(* PLC project Test, Lolitech PLCOpenEditorExample 1.0 *)
(* stored: creationDateTime 2006-09-07 18:52:43 *)

FUNCTION FBDTest : BOOL
  VAR_INPUT
    IN1 : BOOL := false;
    IN2 : BOOL := [4, [0, 1]];
    IN3 : BOOL;
  END_VAR
  VAR  (* added by the conversion: wires and edge detectors of the diagram *)
    R_TRIG1 : R_TRIG;
  END_VAR

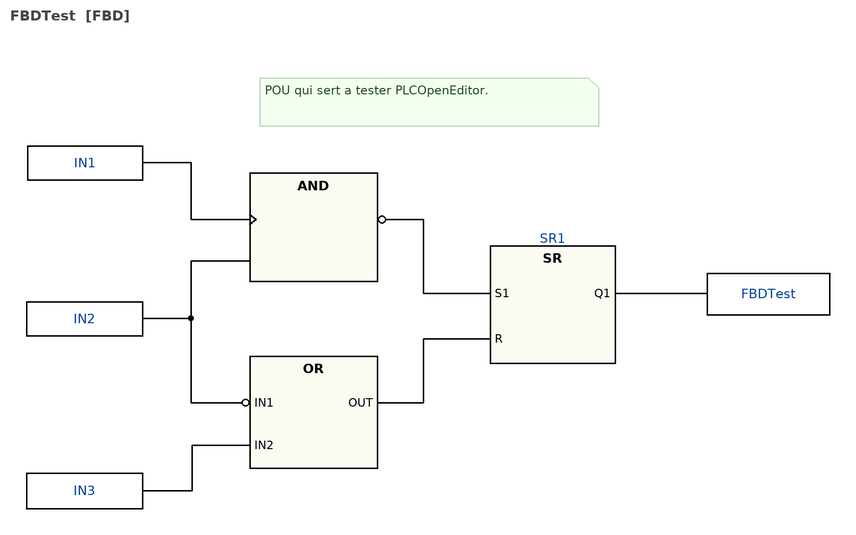
(* FBD diagram, written out as Structured Text *)
(* POU qui sert a tester PLCOpenEditor. *)
R_TRIG1(CLK := IN1);
SR1(S1 := NOT (R_TRIG1.Q AND IN2), R := NOT IN2 OR IN3);
FBDTest := SR1.Q1;
END_FUNCTION

FUNCTION LDTest : BOOL
  VAR_INPUT
    IN1 : BOOL;
    IN2 : BOOL;
    IN3 : BOOL;
    IN4 : BOOL;
  END_VAR

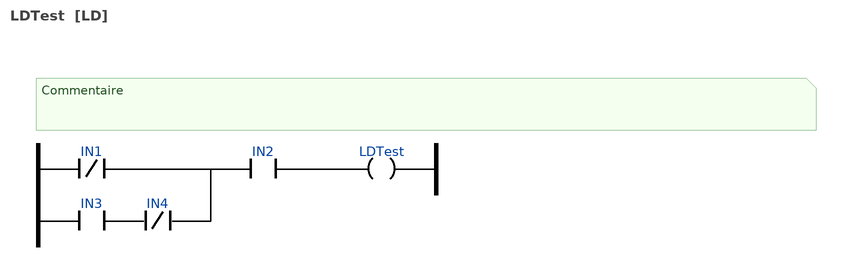
(* LD diagram, written out as Structured Text *)
(* Commentaire *)
LDTest := (NOT IN1 OR IN3 AND NOT IN4) AND IN2;
END_FUNCTION

FUNCTION ILTest : REAL
  VAR_INPUT
    X1 : REAL;
  END_VAR
  VAR
    Temp : REAL;
  END_VAR
  VAR_INPUT
    X2 : REAL;
    Y1 : REAL;
    Y2 : REAL;
    TMax : REAL;
  END_VAR
  VAR_OUTPUT
    ENO : BOOL;
  END_VAR

LD   Y1
SUB  Y2     (* Substract Y2 from Y1 *)
ST   Temp   (* Store Y1-Y2 in Temp *)
MUL  Temp   (* Multiply by Temp to square *)
ADD( X1     (* Defer ADD *)
SUB  X2     (* Substract X1 from X2 *)
ST   Temp   (* Store X1-X2 in Temp *)
MUL  Temp   (* Multiply by Temp to square *)
)
CAL  SQRT   (* Call Square root fun *)
ST   ILTest (* Setup function result *)
GT   TMax   (* Greater than TMax ? *)
JMPC ERR    (* Yes, Jump to Error *)
S    ENO    (* Set ENO *)
RET         (* Normal return *)

ERR:
RET         (* Error return, ENO not set *)
          
END_FUNCTION

PROGRAM SFCTest
  VAR_INPUT
    IN1 : BOOL;
    IN2 : BOOL;
    IN3 : BOOL;
    IN4 : BOOL;
    IN5 : BOOL;
  END_VAR

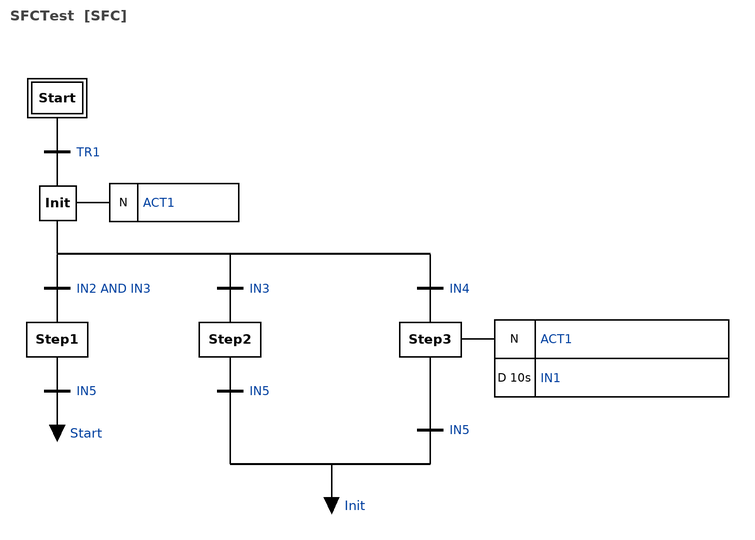
INITIAL_STEP Start:
END_STEP
TRANSITION FROM Start TO Init  (* TR1 *)
  := AND(IN1, IN2, IN3);
END_TRANSITION
STEP Init:
  ACT1(N);
END_STEP
TRANSITION FROM Init TO Step1
  := IN2 AND IN3;
END_TRANSITION
TRANSITION FROM Init TO Step2
  := IN3;
END_TRANSITION
TRANSITION FROM Init TO Step3
  := IN4;
END_TRANSITION
STEP Step1:
END_STEP
TRANSITION FROM Step1 TO Start
  := IN5;
END_TRANSITION
STEP Step2:
END_STEP
TRANSITION FROM Step2 TO Init
  := IN5;
END_TRANSITION
STEP Step3:
  ACT1(N, IN5);
  IN1(D, 10s);
END_STEP
TRANSITION FROM Step3 TO Init
  := IN5;
END_TRANSITION

ACTION ACT1:
IF IN1 THEN
	IN2 := 1;
ELSE
	IN3 := 1;
END_IF;
              
END_ACTION
END_PROGRAM

FUNCTION_BLOCK STTest
  VAR_INPUT
    Collision : BOOL;
    Gate : BOOL;
    Pump : BOOL;
    Temp : INT;
  END_VAR
  VAR_OUTPUT
    Speed : INT;
    PumpSpeed : INT;
    Brakes : BOOL;
    Control_State : BOOL;
  END_VAR

IF Collision THEN
	Speed := 0;
	Brakes := ON;
END_IF;

IF (Gate = CLOSED) AND
		(Pump = ON) AND (Temp > 200.0) THEN
	Control_State := Active;
ELSE
	Control_State := Hold;
	PumpSpeed := 10.0;
END_IF;
          
END_FUNCTION_BLOCK

CONFIGURATION ConfigTest
  VAR_GLOBAL
    Toto AT M10 : INT;
    Tutu AT M20 : BOOL;
  END_VAR
  RESOURCE ResourceTest ON PLC
    VAR_GLOBAL
      Titi AT M30 : INT;
    END_VAR
    TASK Toto(INTERVAL := 10ms, PRIORITY := 6);
    PROGRAM Program1 WITH Toto : SFCTest;
  END_RESOURCE
END_CONFIGURATION

CONFIGURATION ConfigTest2
END_CONFIGURATION
